{attribute addProperty BoxType "EPP6090-0000-0017"}
{attribute addProperty Id "DIS_InputsAT %I*DIS_Inputs_23B85B6E1620DIS_OutputsAT %Q*DIS_Outputs_1C156EA83240WcStateAT %I*WcState_98A4DF7520.250InfoDataAT %I*InfoData_BC63D37F80100"}
{attribute addProperty CRC "1401789242"}
{attribute addProperty SizeInBites "130"}
{attribute addProperty SizeInBytes "16.25"}
TYPE EPP6090_7D66C950 :
STRUCT
	{attribute addProperty Name "DIS_Inputs"}
	DIS_Inputs : DIS_Inputs_23B85B6E;
	{attribute addProperty Name "DIS_Outputs"}
	DIS_Outputs : DIS_Outputs_1C156EA8;
	{attribute addProperty Name "WcState"}
	WcState : WcState_98A4DF75;
	{attribute addProperty Name "InfoData"}
	InfoData : InfoData_BC63D37F;
END_STRUCT
END_TYPE

(* stored: Version 1.2.0.0, ProductVersion 3.1.4024.9
   DUT EPP6090_7D66C950: Id {dc95a0aa-61a3-4ebc-abad-2a71a699c370} *)
